// TwinCAT 3 PLC project LabExercise
// ProgramVersion: 3.1.4023.0
// libraries:
//   Tc2_NCI, * (Beckhoff Automation GmbH)
//   Tc2_Standard, * (Beckhoff Automation GmbH)
//   Tc2_System, * (Beckhoff Automation GmbH)
//   Tc3_Module, * (Beckhoff Automation GmbH)
//   VisuDialogs, * (System)
// project tree:
//   DUTs/ E_Buttons.TcDUT, E_Joystick.TcDUT, E_Light.TcDUT, ST_AnimationScaling.TcDUT (not stored), ST_CraneKinematics.TcDUT (not stored), E_Mode.TcDUT, E_Status.TcDUT, ST_EndStops.TcDUT, ST_Parameters.TcDUT, ST_PistonRange.TcDUT, ST_RelativeMovement.TcDUT (not stored)
//   / GlobalTextList.TcGTLO, PlcTask.TcTTO, Visualization Manager.TcVMO (not stored)
//   GVLs/ HMI.TcGVL, Inputs.TcGVL, Outputs.TcGVL, Parameters.TcGVL
//   Interfaces/ I_Mode.TcIO
//   POUs/ CraneSimulation.TcPOU, MAIN.TcPOU
//   POUs/Function blocks/ FB_ModeControlBox.TcPOU, FB_ModeVisualization.TcPOU, FB_ModeSelector.TcPOU, FB_PositionSimulator.TcPOU, FB_SimulationTime.TcPOU, FB_Softstop.TcPOU, FB_Status.TcPOU
//   POUs/Functions/ F_BarToEng.TcPOU (not stored), F_BoomAnimation.TcPOU (not stored), F_LminToEng.TcPOU (not stored), F_PistonDisplacementToBoomAngle.TcPOU, F_RadToDeg.TcPOU (not stored), F_UpdateParametersByReference.TcPOU
//   VISUs/ CraneHMI.TcVIS
// real-time tasks:
//   TASK PlcTask: cycle T#10ms, priority 20, ADS port 350

CONFIGURATION LabExercise
    RESOURCE PLC ON TwinCAT3
        TASK PlcTask(INTERVAL := T#10ms, PRIORITY := 20);
        PROGRAM MAIN WITH PlcTask : MAIN;
    END_RESOURCE
END_CONFIGURATION

// ---- DUTs/E_Buttons.TcDUT
{attribute 'qualified_only'}
{attribute 'strict'}
TYPE E_Buttons :
(
	Start,
	Stop
);
END_TYPE

// ---- DUTs/E_Joystick.TcDUT
{attribute 'qualified_only'}
{attribute 'strict'}
TYPE E_Joystick :
(
	JoyX,
	JoyY
);
END_TYPE

// ---- DUTs/E_Light.TcDUT
{attribute 'qualified_only'}
{attribute 'strict'}
TYPE E_Light :
(
	green,
	Red
);
END_TYPE

// ---- DUTs/E_Mode.TcDUT
{attribute 'qualified_only'}
{attribute 'strict'}
TYPE E_Mode :
(
	Off := 1,
	Manual,
	Auto
);
END_TYPE

// ---- DUTs/E_Status.TcDUT
{attribute 'qualified_only'}
{attribute 'strict'}
TYPE E_Status :
(
	PowerOff,
	Fault,
	Ready,
	Starting,
	Running,
	Stopping,
	Checking
);
END_TYPE

// ---- DUTs/ST_EndStops.TcDUT
TYPE ST_EndStops :
STRUCT
	sNoEndStop : STRING := 'End Stop not active';
	sPistonUpperEndStop : STRING := 'Piston has reached upper end stop';
	sPistonLowerEndStop : STRING := 'Piston has reached lower end stop';
END_STRUCT
END_TYPE

// ---- DUTs/ST_Parameters.TcDUT
TYPE ST_Parameters :
STRUCT
	fCyclicTime : LREAL := 0.01; 
	stAnimationScaling : ST_AnimationScaling;
	stPistonRange : ST_PistonRange; 
	stCraneKinematics : ST_CraneKinematics;
END_STRUCT
END_TYPE

// ---- DUTs/ST_PistonRange.TcDUT
TYPE ST_PistonRange :
STRUCT
	fPistonPosMin : LREAL :=0;
	fPistonPosMax : LREAL :=0.5;
END_STRUCT
END_TYPE

// ---- GVLs/HMI.TcGVL
{attribute 'qualified_only'}
VAR_GLOBAL
 	fSimulationTime : LREAL; 
	fCylinderVelocityReference : LREAL; 
	fBoomAngleDeg : LREAL;
	fMaxPistonPosition : LREAL;
	sPistonEndStopMessages : STRING;
	bOn : BOOL;
	bAuto : BOOL;
	bPowerOn : BOOL;
	bStart : BOOL;
	bStop : BOOL;
	bRunning : BOOL;
	eMode : E_Mode;
	fManualCylinderPositionReference : LREAL; 
	fCylinderPosition : LREAL; 
	fCylinderPositionRestricted : LREAL; 
	stPistonAnimation : ST_RelativeMovement;
	stBoomAnimation : ST_RelativeMovement;
	eStatus : E_Status;
END_VAR

// ---- GVLs/Inputs.TcGVL
{attribute 'qualified_only'}
VAR_GLOBAL
	bAutoMode : BOOL; 
	bManualMode : BOOL; 
	fJoyY : LREAL;
END_VAR

// ---- GVLs/Outputs.TcGVL
{attribute 'qualified_only'}
VAR_GLOBAL
	fCylinderVelocity : LREAL;
	fCylinderPosition : LREAL;
	bPistonUpperEndStop : BOOL; 
	bPistonLowerEndStop : BOOL; 
	eMode : E_Mode;
END_VAR

// ---- GVLs/Parameters.TcGVL
{attribute 'qualified_only'}
VAR_GLOBAL
	stParam : ST_Parameters;
END_VAR

// ---- Interfaces/I_Mode.TcIO
INTERFACE I_Mode

METHOD Auto
VAR_INPUT
	bEnable : BOOL;
END_VAR
END_METHOD

METHOD Manual
VAR_INPUT
	bEnable : BOOL;
END_VAR
END_METHOD

METHOD Off
VAR_INPUT
	bEnable : BOOL;
END_VAR
END_METHOD

END_INTERFACE

// ---- POUs/MAIN.TcPOU
PROGRAM MAIN
VAR
END_VAR

CraneSimulation();

END_PROGRAM

// ---- POUs/CraneSimulation.TcPOU
PROGRAM CraneSimulation
VAR
	fTime : LREAL; 	
	fPositionAutoMode : LREAL; 
	fInitialPosition : LREAL; 
	fInitialVelocity : LREAL;  
	bPistonMaxNewValue : BOOL;
	fPressureEng : REAL;
	fFlowEng : REAL;
	fPressureBar : LREAL := 60;
	fFlowLmin : LREAL := 20;
	fBoomAngleRad : LREAL;
	fBoomAnimation : LREAL;
	fbModeSelector : FB_ModeSelector;
	fbStatus : FB_Status;
	fbSimulationTime : FB_SimulationTime;
	fbPositionSimulator : FB_PositionSimulator;
END_VAR

// Status
fbStatus(
bPowerOn := HMI.bPowerOn,
bFault := FALSE,
bStart:= HMI.bStart,
bStop := HMI.bStop,
bRunning := HMI.bRunning,
eStatus => HMI.eStatus
);

// Mode Selector
fbModeSelector(bControlBox := FALSE);

// Simulation Time
fbSimulationTime(
eMode := HMI.eMode,
eStatus := HMI.eStatus,
stParam := Parameters.stParam,
fTime => HMI.fSimulationTime
);

// Position Simulation and Animation
IF  HMI.eStatus = E_Status.Ready OR HMI.eStatus = E_Status.Starting OR HMI.eStatus = E_Status.Running THEN
	fbPositionSimulator(
		eMode := HMI.eMode,
		stParam := Parameters.stParam,
		fTime := HMI.fSimulationTime,
		fPositionReference := HMI.fManualCylinderPositionReference,
		fVelocityReference := HMI.fCylinderVelocityReference,
		fInitialVelocity := 0.0,
		fInitialPosition := 0.0,
		bRunning => HMI.bRunning,
		sPistonEndStopMessages => HMI.sPistonEndStopMessages,
		fPositionRestricted => HMI.fCylinderPosition,
		stBoomAnimation => HMI.stBoomAnimation,
		stPistonAnimation => HMI.stPistonAnimation,
		fBoomAngleDeg =>  HMI.fBoomAngleDeg
	);
END_IF

F_UpdateParametersByReference( 
	bSetNewValue := bPistonMaxNewValue,
	fMaxPistonStroke := HMI.fMaxPistonPosition,
	paramCylinderPiston := Parameters.stParam.stPistonRange
);

END_PROGRAM

// ---- POUs/Function blocks/FB_ModeSelector.TcPOU
FUNCTION_BLOCK FB_ModeSelector
VAR_INPUT
	bControlBox : BOOL;
END_VAR
VAR_OUTPUT
END_VAR
VAR
	fbModeVisualization : FB_ModeVisualization;
	fbModeControlBox : FB_ModeControlBox;
	fbMode : I_Mode := fbModeVisualization;
END_VAR

IF NOT(bControlBox) THEN 
	fbMode := fbModeVisualization;
	IF NOT(HMI.bOn) THEN
			fbMode.Off(TRUE); 
			fbMode.Manual(FALSE); 
			fbMode.Auto(FALSE); 
	ELSIF HMI.bOn AND NOT(HMI.bAuto) THEN
			fbMode.Off(FALSE); 
			fbMode.Manual(TRUE); 
			fbMode.Auto(FALSE); 
	ELSIF HMI.bOn AND HMI.bAuto THEN	
			fbMode.Off(FALSE); 
			fbMode.Manual(FALSE); 
			fbMode.Auto(TRUE); 
	ELSE	
			fbMode.Off(FALSE); 
			fbMode.Manual(FALSE); 
			fbMode.Auto(FALSE); 	
	END_IF
	
	
ELSE	  
	fbMode := fbModeControlBox;
	IF NOT(Inputs.bManualMode) AND NOT(Inputs.bAutoMode) THEN
			fbMode.Off(TRUE); 
			fbMode.Manual(FALSE); 
			fbMode.Auto(FALSE); 
	ELSIF Inputs.bManualMode AND NOT(Inputs.bAutoMode) THEN
			fbMode.Off(FALSE); 
			fbMode.Manual(TRUE); 
			fbMode.Auto(FALSE); 
	ELSIF NOT(Inputs.bManualMode) AND Inputs.bAutoMode THEN	
			fbMode.Off(FALSE); 
			fbMode.Manual(FALSE); 
			fbMode.Auto(TRUE); 
	ELSE	
			fbMode.Off(FALSE); 
			fbMode.Manual(FALSE); 
			fbMode.Auto(FALSE); 	
	END_IF
	
END_IF

END_FUNCTION_BLOCK

// ---- POUs/Function blocks/FB_ModeVisualization.TcPOU
FUNCTION_BLOCK PUBLIC FB_ModeVisualization IMPLEMENTS I_Mode
VAR_INPUT
END_VAR
VAR_OUTPUT
END_VAR
VAR
END_VAR

METHOD Auto
VAR_INPUT
	bEnable	: BOOL;
END_VAR
IF bEnable THEN
HMI.fCylinderPosition := CraneSimulation.fPositionAutoMode;
HMI.eMode := E_Mode.Auto; 
END_IF
END_METHOD

METHOD Manual
VAR_INPUT
	bEnable	: BOOL;
END_VAR
IF bEnable THEN
HMI.fCylinderPosition := HMI.fManualCylinderPositionReference;
HMI.eMode := E_Mode.Manual; 
END_IF
END_METHOD

METHOD Off
VAR_INPUT
	bEnable	: BOOL;
END_VAR
IF bEnable THEN
HMI.fCylinderPosition := 0;
HMI.eMode := E_Mode.Off; 
END_IF
END_METHOD

END_FUNCTION_BLOCK

// ---- POUs/Function blocks/FB_ModeControlBox.TcPOU
FUNCTION_BLOCK PUBLIC FB_ModeControlBox IMPLEMENTS I_Mode
VAR_INPUT
END_VAR
VAR_OUTPUT
END_VAR
VAR
END_VAR

METHOD Auto
VAR_INPUT
	bEnable	: BOOL;
END_VAR
IF bEnable THEN
Outputs.fCylinderPosition := CraneSimulation.fPositionAutoMode;
Outputs.eMode := E_Mode.Auto; 
END_IF
END_METHOD

METHOD Manual
VAR_INPUT
	bEnable	: BOOL;
END_VAR
IF bEnable THEN
Outputs.fCylinderPosition := HMI.fManualCylinderPositionReference;
Outputs.eMode := E_Mode.Manual;
END_IF
END_METHOD

METHOD Off
VAR_INPUT
	bEnable	: BOOL;
END_VAR
IF bEnable THEN
Outputs.fCylinderPosition := 0;
Outputs.eMode := E_Mode.Off; 
END_IF
END_METHOD

END_FUNCTION_BLOCK

// ---- POUs/Function blocks/FB_Status.TcPOU
FUNCTION_BLOCK FB_Status
VAR_INPUT
	bPowerOn : BOOL;
	bFault : BOOL;
	bStart : BOOL;
	bStop : BOOL;
	bRunning : BOOL;
END_VAR
VAR_OUTPUT
	eStatus : E_Status := E_Status.Checking;
END_VAR
VAR
END_VAR

CASE eStatus OF 
	E_Status.Checking:
		IF NOT(bFault) THEN
			eStatus := E_Status.Ready;
		ELSE
			eStatus := E_Status.Fault;
		END_IF
		
		IF bPowerOn THEN	
			eStatus := E_Status.Ready;
		ELSE
			eStatus := E_Status.PowerOff;
		END_IF
		
	E_Status.PowerOff:	
		IF bPowerOn THEN	
			eStatus := E_Status.Checking;
		END_IF

	E_Status.Fault:
		IF NOT(bFault) THEN
			eStatus := E_Status.Checking;
		END_IF
	
	E_Status.Ready:
		IF bStart AND bPowerOn AND NOT(bFault) THEN
			eStatus := E_Status.Starting;
		END_IF	
		
		IF  NOT(bPowerOn) OR bFault THEN
			eStatus := E_Status.Checking;
		END_IF	

	E_Status.Starting:
		IF bRunning THEN
			eStatus := E_Status.Running;
		ELSE 
			eStatus := E_Status.Checking;
		END_IF
	
	E_Status.Running:
	
		IF bStop THEN
			eStatus := E_Status.Stopping;
		END_IF
		
		IF NOT(bRunning) OR NOT(bPowerOn) OR bFault THEN
			eStatus := E_Status.Checking;
		END_IF
	
	E_Status.Stopping:	
		IF NOT(bRunning) THEN
			eStatus := E_Status.Checking;
		END_IF
	
		IF bPowerOn OR bFault THEN
		eStatus := E_Status.Checking;
		END_IF	
	
ELSE 	
	eStatus := E_Status.Checking;
END_CASE

END_FUNCTION_BLOCK

// ---- POUs/Function blocks/FB_SimulationTime.TcPOU
FUNCTION_BLOCK FB_SimulationTime
VAR_INPUT
	eStatus : E_Status;
	eMode : E_Mode;
	stParam : ST_Parameters;
END_VAR
VAR_OUTPUT
	fTime : LREAL;
END_VAR
VAR
END_VAR

IF (eStatus = E_Status.Starting OR eStatus = E_Status.Running) AND eMode = E_Mode.Auto  THEN
	fTime := fTime + stParam.fCyclicTime;
ELSE
	fTime := 0; 	
END_IF

END_FUNCTION_BLOCK

// ---- POUs/Function blocks/FB_PositionSimulator.TcPOU
FUNCTION_BLOCK FB_PositionSimulator
VAR_INPUT
	eMode : E_Mode;
	stParam : ST_Parameters;
	fTime : LREAL;
	fPositionReference : LREAL;
	fVelocityReference : LREAL;
	fInitialVelocity : LREAL;
	fInitialPosition : LREAL;
END_VAR
VAR_OUTPUT
	bRunning : BOOL;
	bPistonLowerEndStop : BOOL;
	bPistonUpperEndStop : BOOL;
	sPistonEndStopMessages : STRING; 
	fPositionRestricted : LREAL;
	stBoomAnimation : ST_RelativeMovement;
	stPistonAnimation : ST_RelativeMovement;
	fBoomAngleDeg : LREAL;
END_VAR
VAR
	fPosition : LREAL;
	fbPistonEndStop : FB_Softstop; 
	fBoomAngleRad : LREAL;
	fBoomAnimation : LREAL;
END_VAR

IF  eMode = E_Mode.Manual THEN
	bRunning := FALSE;
	fPosition := fPositionReference;
ELSIF fTime > 0 AND eMode = E_Mode.Auto  THEN 
	bRunning := TRUE;
	fPosition := fVelocityReference * 1/2*(fTime*fTime) + fInitialVelocity * fTime + fInitialPosition;
ELSE
	bRunning := FALSE;
	fPosition := 0.0;
END_IF

// Softstop
fbPistonEndStop(
	fInputValue := fPosition,
	fNegDirLimit := stParam.stPistonRange.fPistonPosMin,
	fPosDirLimit := stParam.stPistonRange.fPistonPosMax,
	bEndStopNegDir => bPistonLowerEndStop,
	bEndStopPosDir => bPistonUpperEndStop,
	sEndStopMessage => sPistonEndStopMessages,
	fOutputValue => fPositionRestricted
);

// Convert Piston Displacement to Boom Angle
fBoomAngleRad := F_PistonDisplacementToBoomAngle(xCyl := fPositionRestricted);
fBoomAngleDeg := F_RadToDeg(fRad := fBoomAngleRad);

// Piston Animation
stPistonAnimation.pt1_y := LREAL_TO_INT(fPositionRestricted * stParam.stAnimationScaling.fPistonScale);

// Boom Animation
fBoomAnimation := F_BoomAnimation(
	fScale := stParam.stAnimationScaling.fBoomScale,
	fBoomAngle := fBoomAngleRad,
	fBoomLength := stParam.stCraneKinematics.fBoomLength,
	fBoomTipX => stBoomAnimation.pt1_x,
	fBoomTipY => stBoomAnimation.pt1_y
);

END_FUNCTION_BLOCK

// ---- POUs/Function blocks/FB_Softstop.TcPOU
FUNCTION_BLOCK FB_Softstop
VAR_INPUT
	fInputValue : LREAL;
	fNegDirLimit : LREAL;
	fPosDirLimit : LREAL;
END_VAR
VAR_OUTPUT
	bEndStopNegDir : BOOL;
	bEndStopPosDir : BOOL;
	sEndStopMessage : STRING;
	fOutputValue : LREAL;
END_VAR
VAR
	aEndStopMessages : ARRAY [0..2] OF STRING := ['EndStop not active','EndStop Negative Direction Active','EndStop Positive Direction Active'];
END_VAR

IF fInputValue <= fNegDirLimit THEN 
	bEndStopNegDir := TRUE; 
	bEndStopPosDir := FALSE; 
	sEndStopMessage := aEndStopMessages[1];
	fOutputValue := fNegDirLimit;
ELSIF fInputValue >= fPosDirLimit THEN 
	bEndStopNegDir := FALSE; 
	bEndStopPosDir := TRUE; 
	sEndStopMessage := aEndStopMessages[2];
	fOutputValue := fPosDirLimit;
ELSE 
	bEndStopNegDir := FALSE; 	
	bEndStopPosDir := FALSE; 	
	sEndStopMessage := aEndStopMessages[0];
	fOutputValue := fInputValue;
END_IF

END_FUNCTION_BLOCK

// ---- POUs/Functions/F_PistonDisplacementToBoomAngle.TcPOU
FUNCTION F_PistonDisplacementToBoomAngle : LREAL
VAR_INPUT
	xCyl : LREAL;
END_VAR
VAR
	AB : LREAL;
	AC : LREAL;
	BC : LREAL;
	alpha1 : LREAL;
	alpha2 : LREAL;
	theta1 : LREAL;
	AB2 : LREAL;
	AC2 : LREAL;
	BC2 : LREAL;
END_VAR

AB := SQRT(ABS(Parameters.stParam.stCraneKinematics.ABx)*ABS(Parameters.stParam.stCraneKinematics.ABx) + ABS(Parameters.stParam.stCraneKinematics.ABy)*ABS(Parameters.stParam.stCraneKinematics.ABy));
AC := SQRT(ABS(Parameters.stParam.stCraneKinematics.ACx)*ABS(Parameters.stParam.stCraneKinematics.ACx) + ABS(Parameters.stParam.stCraneKinematics.ACy)*ABS(Parameters.stParam.stCraneKinematics.ACy));

BC := 0.77222 + xCyl;

alpha1 := ATAN(ABS(Parameters.stParam.stCraneKinematics.ACy)/ ABS(Parameters.stParam.stCraneKinematics.ACx));
alpha2 := ATAN(ABS(Parameters.stParam.stCraneKinematics.ABy)/ ABS(Parameters.stParam.stCraneKinematics.ABx));

AB2 := ABS(AB)*ABS(AB);
AC2 := ABS(AC)*ABS(AC);
BC2 := ABS(BC)*ABS(BC);

theta1 := ACOS( (AB2 + AC2 - BC2) / (2 * ABS(AB) * ABS(AC)) ) - alpha2 + alpha1;

F_PistonDisplacementToBoomAngle := theta1;

END_FUNCTION

// ---- POUs/Functions/F_UpdateParametersByReference.TcPOU
FUNCTION F_UpdateParametersByReference 
VAR_INPUT
	bSetNewValue : BOOL;
	fMaxPistonStroke : LREAL;
	paramCylinderPiston : REFERENCE TO ST_PistonRange;
END_VAR
VAR

END_VAR

IF bSetNewValue THEN
	paramCylinderPiston.fPistonPosMax := fMaxPistonStroke;
	bSetNewValue := FALSE;
END_IF

END_FUNCTION

// ---- GlobalTextList.TcGTLO
TEXTLIST GlobalTextList
  624 = '%0.1f'
  198 = '%f'
  949 = '%i'
  819 = '%s'
  850 = '%s '
  935 = '0.5m'
  892 = '0m'
  807 = '1m'
  948 = '1mx0'
  175 = 'AUTO'
  104 = 'Boom Angle: %0.1f [deg]'
  236 = 'Clock: %s [s]'
  58 = 'Current Max Piston Stroke: %0.1f [m] '
  471 = 'Cylinder Position Reference: %0.1f [m]'
  995 = 'Cylinder Position Reference: %f [m]'
  752 = 'Cylinder Velocity Reference: %0.0001f [m/s]'
  954 = 'Cylinder Velocity Reference: %0.01f [m/s]'
  105 = 'Cylinder Velocity Reference: %0.1f [m/s]'
  755 = 'Cylinder Velocity Reference: %0.1s [m/s]'
  25 = 'Cylinder Velocity Reference: %f [m/s]'
  308 = 'Cylinder Velocity Reference: %f [m]'
  30 = 'Cylinder Velocity Reference: %i'
  903 = 'Cylinder Velocity Reference: %s'
  128 = 'Cylinder Velocity Reference: %s [m/s]'
  353 = 'Enable'
  409 = 'ENABLE'
  527 = 'End Stop Status: %s '
  660 = 'MANUAL'
  8 = 'Manual Cylinder Position   Reference [m]'
  157 = 'Manual Cylinder Position Reference'
  7 = 'Max Piston Stroke: %0.1f [m] '
  110 = 'Max Piston Stroke: %f [m] '
  84 = 'Max Stroke: %f [m] '
  188 = 'Mode'
  76 = 'Mode: %s '
  646 = 'New Max Piston Stroke: %0.1f [m] '
  65 = 'OFF'
  629 = 'ON'
  310 = 'RUNNING'
  695 = 'Set New Value'
  466 = 'Simulation'
  279 = 'Start'
  868 = 'START'
  254 = 'START AUTO'
  978 = 'Started'
  173 = 'Status: %s '
  397 = 'STOP'
  495 = 'Time: %0.1f [s]'
  221 = 'Time: %f [s]'
  61 = 'Time: %i [s]'
  725 = 'Time: %s [s]'
  444 = 'x0'
END_TEXTLIST

// ---- VISUs/CraneHMI.TcVIS
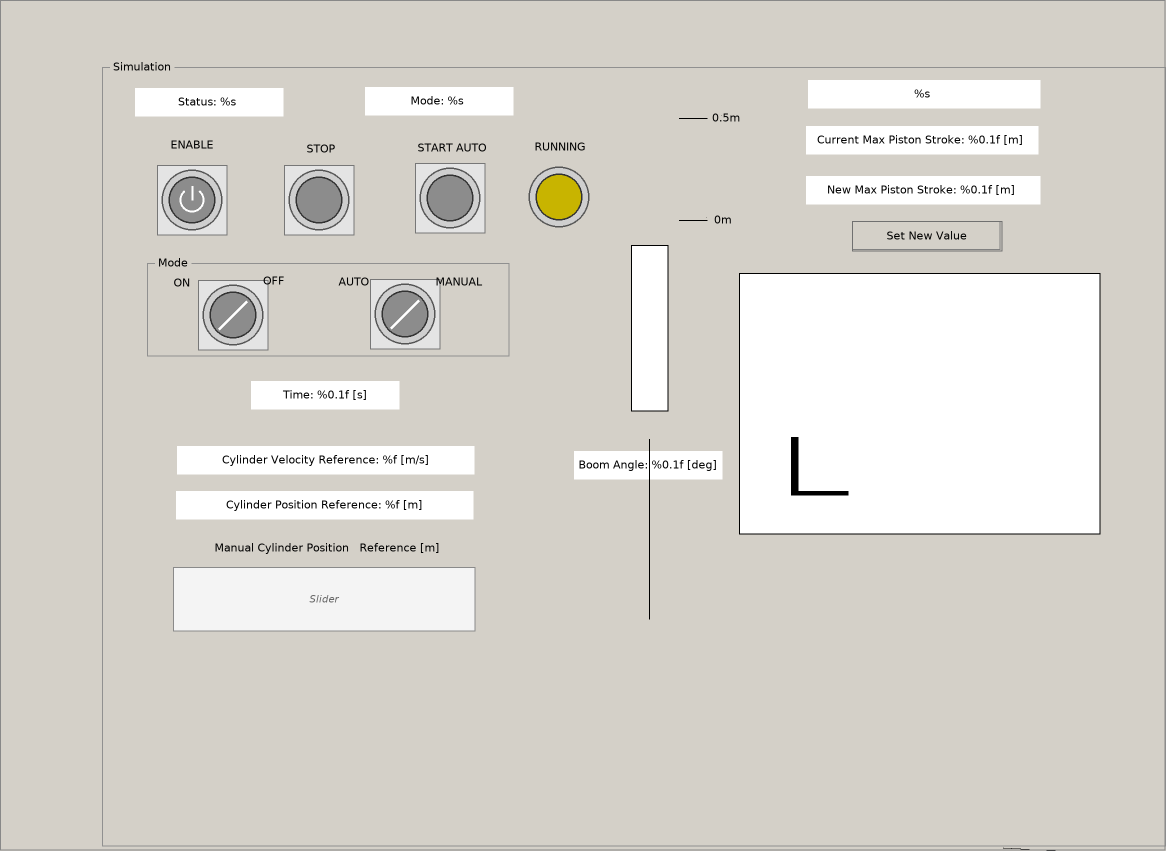
VISUALIZATION CraneHMI  // 1166x851
    Rectangle (566,310 166x37), angle 270
    GroupBox (102,59 1064x787), "Simulation"
        GroupBox (45,196 362x101), "Mode"
        Rectangle (637,214 361x261)
        PowerSwitch (55,106 70x70), variable: HMI.bPowerOn, behaviour: TOGGLE, style: Switch-PowerSwitch-Gray
        PushSwitch (313,104 70x70), variable: HMI.bStart, behaviour: TAP, style: Switch-PushSwitch-Gray
        Lamp1 (422,103 70x70), variable: HMI.bRunning, style: Lamp-Lamp1-Yellow
        Textfield (74,386 299x30), "Cylinder Velocity Reference: %f [m/s]", text variable: HMI.fCylinderVelocityReference
            OnMouseClick: write the text variable via Default
        Label (15,71 150x30), "ENABLE"
        Label (275,74 150x30), "START AUTO"
        Label (383,73 150x30), "RUNNING"
        Textfield (148,321 150x30), "Time: %0.1f [s]", text variable: HMI.fSimulationTime
        Label (90,474 270x30), "Manual Cylinder Position Reference [m]"
        Textfield (73,431 299x30), "Cylinder Position Reference: %f [m]", text variable: HMI.fCylinderPosition
        Line (577,161) (605,161)
        Label (607,146 28x30), "0m"
        Textfield (703,66 234x30), "Current Max Piston Stroke: %0.1f [m]", text variable: Parameters.stParam.stPistonRange.fPistonPosMax
        Textfield (703,116 236x30), "New Max Piston Stroke: %0.1f [m]", text variable: HMI.fMaxPistonPosition
            OnMouseDown: write the text variable via Default, min 0, max 1
        Button (750,162 150x30), "Set New Value"
            tap CraneSimulation.bPistonMaxNewValue
        Line (577,59) (605,59)
        Textfield (32,28 150x30), "Status: %s", text variable: HMI.eStatus
        Textfield (262,27 150x30), "Mode: %s", text variable: HMI.eMode
        Textfield (705,20 234x30), "%s", text variable: HMI.sPistonEndStopMessages
        Textfield (471,391 150x30), "Boom Angle: %0.1f [deg]", text variable: HMI.fBoomAngleDeg
        Slider (71,508 302x64), variable: HMI.fManualCylinderPositionReference, scale 0..0.5
        Rectangle (689,378 7x58)
        Rectangle (690,432 56x4)
        RotarySwitch (96,221 70x70), variable: HMI.bOn, behaviour: TOGGLE, style: Switch-RotarySwitch-Gray
        RotarySwitch (268,220 70x70), variable: HMI.bAuto, behaviour: TOGGLE, style: Switch-RotarySwitch-Gray
        Label (282,208 150x30), "MANUAL"
        Label (177,208 150x30), "AUTO"
        Label (97,207 150x30), "OFF"
        PushSwitch (182,106 70x70), variable: HMI.bStop, behaviour: TAP, style: Switch-PushSwitch-Gray
        Label (144,75 150x30), "STOP"
    Line (649,439) (649,619)
        p1126004900: HMI.stPistonAnimation.pt1_y
        p3528305787: HMI.stPistonAnimation.pt0_x
        p2773130477: HMI.stPistonAnimation.pt0_y
        p874137650: HMI.stPistonAnimation.pt1_x
    Line (706,217) (706,217)
    Label (712,103 28x30), "0.5m"
    Line (721,115) (721,115)
    Line (1055,851) (1003,848)
        p1126004900: HMI.stBoomAnimation.pt1_y
        p3528305787: HMI.stBoomAnimation.pt0_x
        p2773130477: HMI.stBoomAnimation.pt0_y
        p874137650: -HMI.stBoomAnimation.pt1_x
    Label (107,268 150x30), "ON"
END_VISUALIZATION
